// SIMATIC S7-200 SMART project (STEP 7-Micro/WIN SMART), CPU SR20

SYMBOL_TABLE 系统符号
Always_On        SM0.0    // 始终接通
First_Scan_On    SM0.1    // 仅在第一个扫描周期时接通
END_SYMBOL_TABLE

ORGANIZATION_BLOCK MAIN:OB1
TITLE=读液位高度
BEGIN
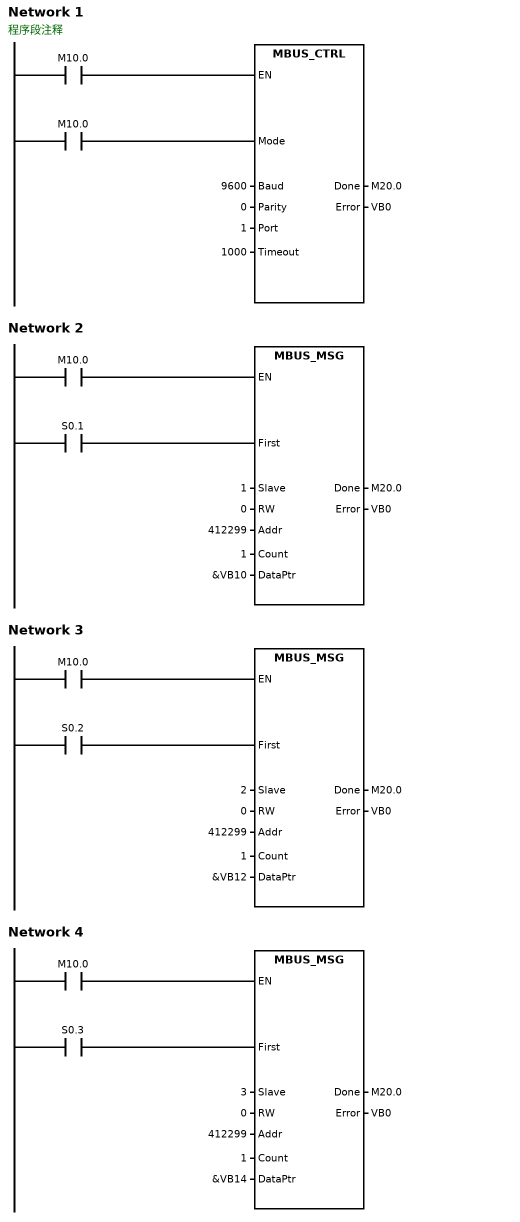
Network 1
// 程序段注释
LD     M10.0
=      L60.0
LD     M10.0
=      L63.7
LD     L60.0
CALL   MBUS_CTRL:SBR1, L63.7, 9600, 0, 1, 1000, M20.0, VB0
Network 2
LD     M10.0
=      L60.0
LD     S0.1
=      L63.7
LD     L60.0
CALL   MBUS_MSG:SBR2, L63.7, 1, 0, 412299, 1, &VB10, M20.0, VB0
Network 3
LD     M10.0
=      L60.0
LD     S0.2
=      L63.7
LD     L60.0
CALL   MBUS_MSG:SBR2, L63.7, 2, 0, 412299, 1, &VB12, M20.0, VB0
Network 4
LD     M10.0
=      L60.0
LD     S0.3
=      L63.7
LD     L60.0
CALL   MBUS_MSG:SBR2, L63.7, 3, 0, 412299, 1, &VB14, M20.0, VB0
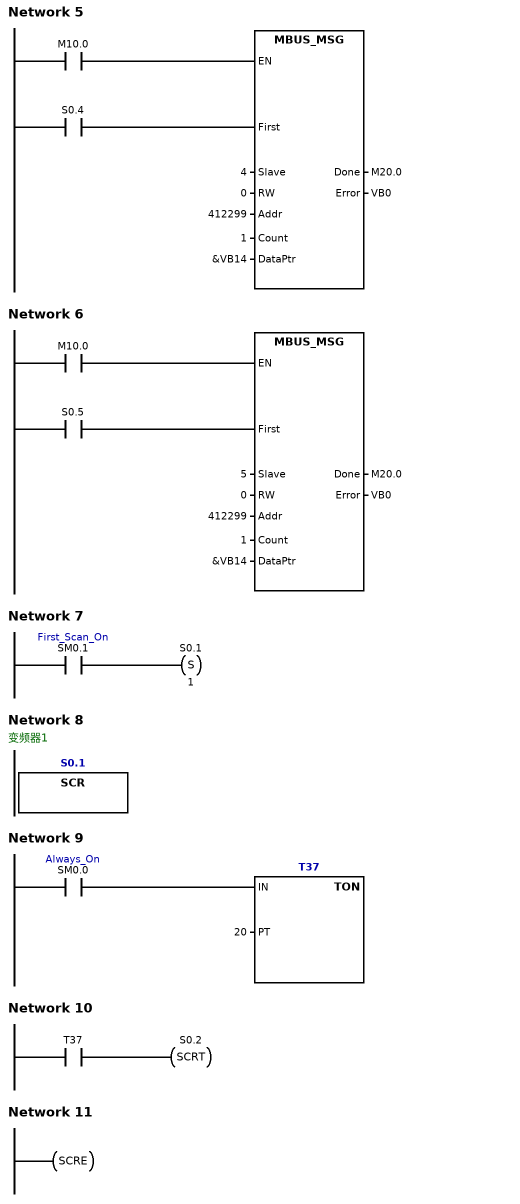
Network 5
LD     M10.0
=      L60.0
LD     S0.4
=      L63.7
LD     L60.0
CALL   MBUS_MSG:SBR2, L63.7, 4, 0, 412299, 1, &VB14, M20.0, VB0
Network 6
LD     M10.0
=      L60.0
LD     S0.5
=      L63.7
LD     L60.0
CALL   MBUS_MSG:SBR2, L63.7, 5, 0, 412299, 1, &VB14, M20.0, VB0
Network 7
LD     First_Scan_On:SM0.1
S      S0.1, 1
Network 8
// 变频器1
LSCR   S0.1
Network 9
LD     Always_On:SM0.0
TON    T37, 20
Network 10
LD     T37
SCRT   S0.2
Network 11
SCRE
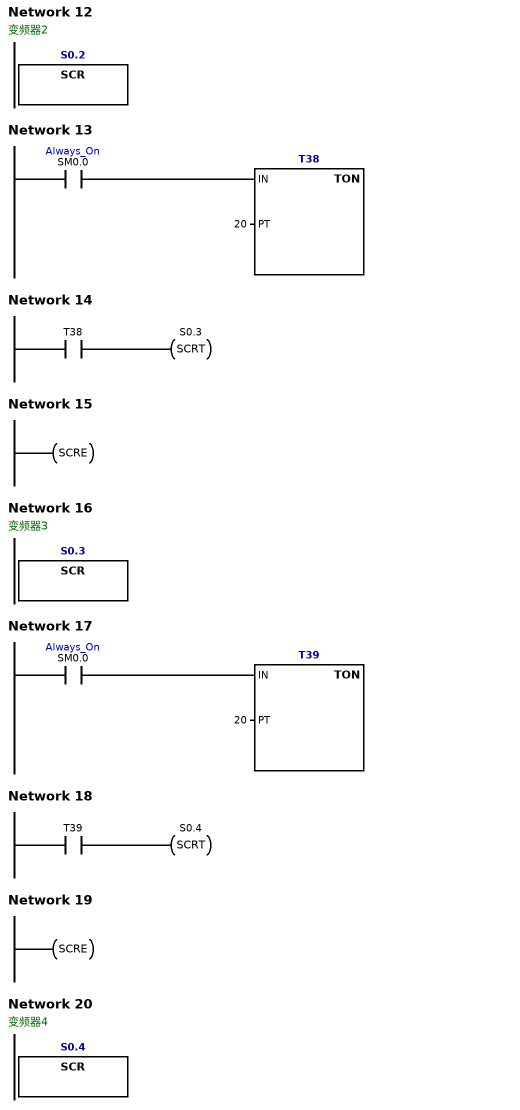
Network 12
// 变频器2
LSCR   S0.2
Network 13
LD     Always_On:SM0.0
TON    T38, 20
Network 14
LD     T38
SCRT   S0.3
Network 15
SCRE
Network 16
// 变频器3
LSCR   S0.3
Network 17
LD     Always_On:SM0.0
TON    T39, 20
Network 18
LD     T39
SCRT   S0.4
Network 19
SCRE
Network 20
// 变频器4
LSCR   S0.4
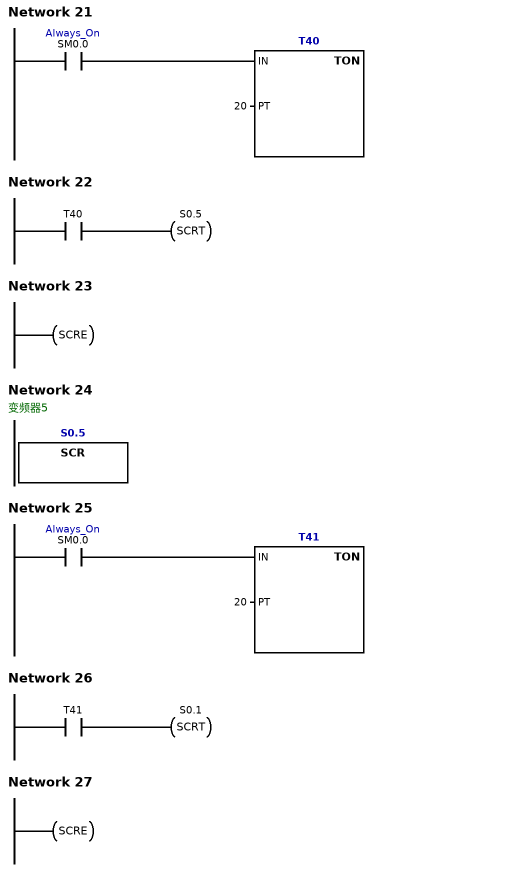
Network 21
LD     Always_On:SM0.0
TON    T40, 20
Network 22
LD     T40
SCRT   S0.5
Network 23
SCRE
Network 24
// 变频器5
LSCR   S0.5
Network 25
LD     Always_On:SM0.0
TON    T41, 20
Network 26
LD     T41
SCRT   S0.1
Network 27
SCRE
Network 34
// 程序段注释
END_ORGANIZATION_BLOCK

// SBR1: protected block, not included

// SBR2: protected block, not included

// SBR3: protected block, not included
